TYPE E_Typ_JUN :
(
	Max_E_Typ_JUN
);
END_TYPE

(* stored: Version 1.1.0.1, ProductVersion 3.1.0.23
   DUT E_Typ_JUN: Id {ef04182f-dde3-4089-94fa-5d27c3bb101d} *)
